(* IEC 61131-3 sources: Std_PalletMover/Class/_JSONWriter (part 2) *)

END_FUNCTION

FUNCTION GLOBAL _JSONWriter::Minify
	VAR_INPUT
		json 	: ^CHAR;
	END_VAR

  _cJSON.Minify(json := json);

END_FUNCTION

FUNCTION GLOBAL _JSONWriter::AddNullToObject
	VAR_INPUT
		object 	: ^_cJSON::t_s_cJSON;
		name 	: ^CHAR;
	END_VAR
	VAR_OUTPUT
		item 	: ^_cJSON::t_s_cJSON;
	END_VAR

  item := _cJSON.AddNullToObject(object  :=  object,
                                name    :=  name);

END_FUNCTION

FUNCTION GLOBAL _JSONWriter::AddTrueToObject
	VAR_INPUT
		object 	: ^_cJSON::t_s_cJSON;
		name 	: ^CHAR;
	END_VAR
	VAR_OUTPUT
		item 	: ^_cJSON::t_s_cJSON;
	END_VAR

  item := _cJSON.AddTrueToObject(object  :=  object,
                                name    :=  name);

END_FUNCTION

FUNCTION GLOBAL _JSONWriter::AddFalseToObject
	VAR_INPUT
		object 	: ^_cJSON::t_s_cJSON;
		name 	: ^CHAR;
	END_VAR
	VAR_OUTPUT
		item 	: ^_cJSON::t_s_cJSON;
	END_VAR

  item := _cJSON.AddFalseToObject( object  :=  object,
                                  name    :=  name);

END_FUNCTION

FUNCTION GLOBAL _JSONWriter::AddBoolToObject
	VAR_INPUT
		object 	: ^_cJSON::t_s_cJSON;
		name 	: ^CHAR;
		boolean 	: BOOL;
	END_VAR
	VAR_OUTPUT
		item 	: ^_cJSON::t_s_cJSON;
	END_VAR

  item := _cJSON.AddBoolToObject(object  :=  object,
                                name    :=  name,
                                boolean :=  boolean);

END_FUNCTION

FUNCTION GLOBAL _JSONWriter::AddNumberToObject
	VAR_INPUT
		object 	: ^_cJSON::t_s_cJSON;
		name 	: ^CHAR;
		number 	: LREAL;
	END_VAR
	VAR_OUTPUT
		item 	: ^_cJSON::t_s_cJSON;
	END_VAR

  item := _cJSON.AddNumberToObject(object  :=  object,
                                  name    :=  name,
                                  number  :=  number);

END_FUNCTION

FUNCTION GLOBAL _JSONWriter::AddStringToObject
	VAR_INPUT
		object 	: ^_cJSON::t_s_cJSON;
		name 	: ^CHAR;
		string 	: ^CHAR;
	END_VAR
	VAR_OUTPUT
		item 	: ^_cJSON::t_s_cJSON;
	END_VAR

  item := _cJSON.AddStringToObject(object  :=  object,
                                  name    :=  name,
                                  string  :=  string);

END_FUNCTION

FUNCTION GLOBAL _JSONWriter::AddRawToObject
	VAR_INPUT
		object 	: ^_cJSON::t_s_cJSON;
		name 	: ^CHAR;
		raw 	: ^CHAR;
	END_VAR
	VAR_OUTPUT
		item 	: ^_cJSON::t_s_cJSON;
	END_VAR

  item := _cJSON.AddRawToObject( object  :=  object,
                                name    :=  name,
                                raw     :=  raw);

END_FUNCTION

FUNCTION GLOBAL _JSONWriter::AddObjectToObject
	VAR_INPUT
		object 	: ^_cJSON::t_s_cJSON;
		name 	: ^CHAR;
	END_VAR
	VAR_OUTPUT
		item 	: ^_cJSON::t_s_cJSON;
	END_VAR

  item := _cJSON.AddObjectToObject(object  :=  object,
                                  name    :=  name);

END_FUNCTION

FUNCTION GLOBAL _JSONWriter::AddArrayToObject
	VAR_INPUT
		object 	: ^_cJSON::t_s_cJSON;
		name 	: ^CHAR;
	END_VAR
	VAR_OUTPUT
		item 	: ^_cJSON::t_s_cJSON;
	END_VAR

  item := _cJSON.AddArrayToObject( object  :=  object,
                                  name    :=  name);

END_FUNCTION

FUNCTION GLOBAL _JSONWriter::SetNumber
	VAR_INPUT
		object 	: ^_cJSON::t_s_cJSON;
		number 	: LREAL;
	END_VAR
	VAR_OUTPUT
		retVal 	: LREAL;
	END_VAR

  retVal := _cJSON.SetNumber(object  :=  object,
                             number  :=  number);

END_FUNCTION

FUNCTION GLOBAL _JSONWriter::SetValuestring
	VAR_INPUT
		object 	: ^_cJSON::t_s_cJSON;
		valueString 	: ^CHAR;
	END_VAR
	VAR_OUTPUT
		retVal 	: ^CHAR;
	END_VAR

  retVal := _cJSON.SetValuestring( object      :=  object,
                                  valueString :=  valueString);

END_FUNCTION

FUNCTION VIRTUAL GLOBAL _JSONWriter::Init

  if _FirstScan then

    ResetMem();
    ClearMainElement();

  end_if;

END_FUNCTION

FUNCTION GLOBAL _JSONWriter::ClearMainElement

  if MainElement <> NIL then
    _cJSON.Delete(item := MainElement);
  end_if;
  MainElement := _cJSON.CreateObject();

END_FUNCTION
